FUNCTION_BLOCK FB_Tree_IndexBased IMPLEMENTS ITF_Tree_IndexBased
VAR_IN_OUT
	a_stNodes : ARRAY[0..63] OF ST_Tree_IndexBased_Node;
END_VAR
VAR_INPUT
	sHead : STRING;
END_VAR
VAR
	bInitialized 	: BOOL;
	nNodeCount 		: DINT;
	nNewNodeIndex	: DINT;
	nHeadIndex		: DINT;
	
	//"Temp" variables for use in AddNodeAsChildByName
	nParentIndex 	: DINT;
	nChildCount		: DINT;
END_VAR

IF NOT bInitialized THEN
	initialize();
END_IF

METHOD AddNodeAsChildByName : BOOL
VAR_INPUT
	sNewName 	: STRING;
	sParentName	: STRING;
END_VAR
nParentIndex := GetIndexByName(sParentName);		//Find the index value of the designated parent node
nChildCount := a_stNodes[nParentIndex].nChildCount;
IF nParentIndex >= 0 THEN	//If GetIndex was successful
	IF (a_stNodes[nParentIndex].nChildCount < 64) THEN	//TODO: Proper Constant bound definition	//If the parent is not at max child count
		a_stNodes[nNewNodeIndex].sName := sNewName;		//assign new node name to next empty node in list
		a_stNodes[nNewNodeIndex].nParent := nParentIndex;	//assign the parent node to the new child node
		a_stNodes[nNewNodeIndex].nDepth := a_stNodes[nParentIndex].nDepth + 1;
		a_stNodes[nParentIndex].a_nChildren[nChildCount] := nNewNodeIndex;		//assign the new node location as the next child in the parent
		nNewNodeIndex := nNewNodeIndex + 1;		//Increment to next empty node
		a_stNodes[nParentIndex].nChildCount := nChildCount + 1;
	END_IF
END_IF
END_METHOD

METHOD GetIndexByName : DINT
VAR_INPUT
	sName : STRING;
END_VAR
VAR
	i : DINT;
END_VAR
FOR i := 0 TO nNodeCount DO
	IF a_stNodes[i].sName = sName THEN
		GetIndexByName := i;
		RETURN;
	END_IF
END_FOR

GetIndexByName := -1;
END_METHOD

METHOD PRIVATE initialize : BOOL
VAR_INPUT
END_VAR
//nNodeCount := UPPER_BOUND(a_stNodes,1) - LOWER_BOUND(a_stNodes,1) + 1;
nNodeCount := 64;
IF nNodeCount >= 0 THEN
	nHeadIndex := 0;//LOWER_BOUND(a_stNodes,1);
	a_stNodes[nHeadIndex].sName := sHead;
	a_stNodes[nHeadIndex].nDepth := 0;
	a_stNodes[nHeadIndex].nParent := -1;
	nNewNodeIndex := nHeadIndex + 1;
END_IF
END_METHOD

END_FUNCTION_BLOCK

(* stored: Version 1.1.0.1, ProductVersion 3.1.4024.9
   POU FB_Tree_IndexBased: Id {329a32fd-f238-4137-9397-ea1d78854c9d}, SpecialFunc None
   Folder 01_ITF_Tree_IndexBased: Id {a3bc00ea-a8f6-421c-938a-2a78cd275621}
   Method AddNodeAsChildByName: Id {cf8f65b6-5cf8-45a5-99be-5fee703fb657}
   Method GetIndexByName: Id {be420560-9e63-430e-939f-9883ff395b2f}
   Method initialize: Id {1c1868c4-1b6a-4140-b4e0-9a7a111582f2} *)
